TYPE U_TRANSLATE_REGS_IN :
UNION
	nArray :	ARRAY [0..31] OF WORD;
	Label : 	S_REGS_IN;
END_UNION
END_TYPE

(* stored: Version 1.1.0.1, ProductVersion 3.1.4024.6
   DUT U_TRANSLATE_REGS_IN: Id {93739cbb-38e6-44be-ad93-d5f80d6ff126} *)
